(* Logix 5000 project; controller Ex_2_09 Emulate 5570 rev 33.11; software revision 33.00 *)
// Turn on lamp tower with a rotary switch

TASK MainTask (continuous, watchdog 500 ms) : MainProgram

MODULES
   Local : Emulate 5570 (ICP 4, rev 33.11)
END_MODULES

VAR_GLOBAL   (* controller tags *)
   P1 : BOOL;   // Lamp P1
   P2 : BOOL;   // Lamp P2
   P3 : BOOL;   // Lamp P3
   S0 : BOOL := 1;   // Setting 0
   S1 : BOOL;   // Setting S1
   S2 : BOOL;   // Setting S2
   S3 : BOOL;   // Setting S3
END_VAR

PROGRAM MainProgram   (* main routine MainRoutine *)

ROUTINE MainRoutine   (* ladder *)
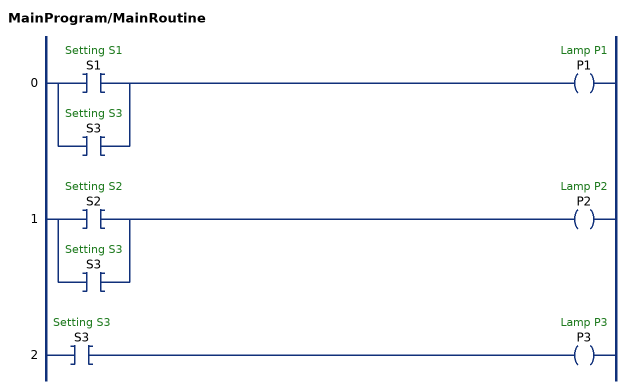
   0: [XIC(S1) ,XIC(S3) ]OTE(P1);
   1: [XIC(S2) ,XIC(S3) ]OTE(P2);
   2: XIC(S3)OTE(P3);
END_ROUTINE
END_PROGRAM
